Staubli VAL3: kill.pgx

public program kill(num x_nConvNum)
begin
  call enc:kill()
  taskKill(sTASK[0]+toString("",x_nConvNum))
  call det:kill()
end
